// Mitsubishi GX Works2 project: 231003-003- exercicios   PLC: Q03UDV

// task Task_01 (event TRUE, interval 0, priority 31): POU_01

PROGRAM POU_01
VAR
  fbBlinker_teste : fbBlinker;
END_VAR
(* structured ladder/FBD written out as ST: instructions are called as NAME(EN, inputs, outputs); _pN, _eN, _tN stand for wires *)
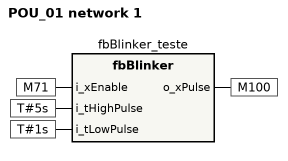
(* network 1 *)
fbBlinker_teste(i_xEnable := M71, i_tHighPulse := T#5s, i_tLowPulse := T#1s, o_xPulse => M100);
END_PROGRAM

FUNCTION_BLOCK fbBlinker
VAR_INPUT
  i_xEnable : BOOL;
  i_tHighPulse : TIME;
  i_tLowPulse : TIME;
END_VAR
VAR_OUTPUT
  o_xPulse : BOOL;
END_VAR
VAR
  fbTimerhigh : TP;
  fbTimerLow : TOF;
  xAuxiliar : BOOL;
  TP_1 : TP;
END_VAR
(* structured ladder/FBD written out as ST: instructions are called as NAME(EN, inputs, outputs); _pN, _eN, _tN stand for wires *)
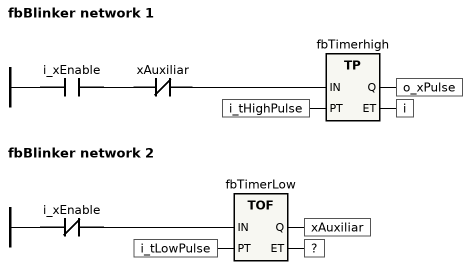
(* network 1 *)
fbTimerhigh(IN := i_xEnable AND NOT xAuxiliar, PT := i_tHighPulse, Q => o_xPulse, ET => i);
(* network 2 *)
fbTimerLow(IN := NOT i_xEnable, PT := i_tLowPulse, Q => xAuxiliar, ET => ?);
END_FUNCTION_BLOCK
